THIS^.resetCycleManager();
configScope := THIS^.cycleManager.configuration;
THIS^.cycleManager.update(execute := TRUE);
AssertEquals_DINT(
	Expected := CNM_ReturnTypes.DefaultSteps.STEP.INIT,
	Actual := THIS^.cycleManager.step.current,
	Message := 'step should be INIT step'
);
// set global stepWidth
configScope.sequence.stepWidth := 7;
THIS^.cycleManager.proceed();
THIS^.cycleManager.update(execute := TRUE);
AssertEquals_DINT(
	Expected := (CNM_ReturnTypes.DefaultSteps.STEP.INIT + 7),
	Actual := THIS^.cycleManager.step.current,
	Message := 'step should be INIT step + 7'
);
// test it twice to make it nice
THIS^.cycleManager.proceed();
THIS^.cycleManager.update(execute := TRUE);
AssertEquals_DINT(
	Expected := (CNM_ReturnTypes.DefaultSteps.STEP.INIT + 14),
	Actual := THIS^.cycleManager.step.current,
	Message := 'step should be INIT step + 14'
);
// proceed with local stepWidth
THIS^.cycleManager.proceedWith(10);
THIS^.cycleManager.update(execute := TRUE);
AssertEquals_DINT(
	Expected := 10,
	Actual := THIS^.cycleManager.step.current,
	Message := 'stepWidth should be ignored by proceedWith(), step should be 10'
);
configScope.step.stepWidth := 5;
THIS^.cycleManager.proceed();
THIS^.cycleManager.update(execute := TRUE);
AssertEquals_DINT(
	Expected := 15,
	Actual := THIS^.cycleManager.step.current,
	Message := 'step should be 15'
);
// proceed again with global stepWidth
THIS^.cycleManager.proceed();
THIS^.cycleManager.update(execute := TRUE);
AssertEquals_DINT(
	Expected := 22,
	Actual := THIS^.cycleManager.step.current,
	Message := 'step should be 22'
);

TcUnit.TEST_FINISHED();
END_METHOD

(*

short summary
=================
Tests different stop request modes.
Verifies AFTER_SUCCESS, AFTER_NOT_SUCCESS, ALWAYS, and IGNORE modes work correctly.

.. <legal notes>

legal notes
=================
| SPDX-FileCopyrightText: © 2025 ekvip automation GmbH <info@ekvip.de>
| SPDX-License-Identifier: Apache-2.0
| For details check: Apache-2.0_

.. _Apache-2.0: https://www.apache.org/licenses/LICENSE-2.0

.. </legal notes>

*)
METHOD PRIVATE testStopRequestModes
VAR_INST
	testState : INT;
END_VAR
RETURN( THIS^.testSuiteAborted OR_ELSE  NOT TcUnit.TEST_ORDERED(THIS^.getTestNameFor('testStopRequestModes')));

CASE testState OF
0: // Initialize
	THIS^.resetCycleManager();
	iConfiguration := cycleManager;
	iCycleManager := cycleManager;
	testState := 10;
	
10: // Test AFTER_SUCCESS mode
	cycleManager.update(execute := TRUE, stopRequest := FALSE);
	
	// Configure stop request mode
	iConfiguration.configuration.sequence.stopRequest.afterSuccessfulStep();
	
	iCycleManager.proceedWith(10);
	cycleManager.update(execute := TRUE, stopRequest := FALSE);
	testState := 20;
	
20: // Evaluate success with stop request
	cycleManager.update(execute := TRUE, stopRequest := TRUE);
	AssertEquals_DINT(
		Expected := 10,
		Actual := iCycleManager.step.current,
		Message := 'Should stay in step 10 until successful evaluate'
	);
	IF iCycleManager.executeStep THEN
		// Evaluate success
		iCycleManager.evaluate(CNM_ReturnTypes.SingleExecutionState.SUCCESS);
		testState := 30;
	END_IF
	
30: // Verify moved to success due to stop request
	cycleManager.update(execute := TRUE, stopRequest := TRUE);
	
	AssertEquals_DINT(
		Expected := CNM_ReturnTypes.DefaultSteps.STEP.SUCCESS,
		Actual := iCycleManager.step.current,
		Message := 'Should move to SUCCESS with stop request after success'
	);
	
	AssertEquals_INT(
		Expected := CNM_ReturnTypes.SingleExecutionState.SUCCESS,
		Actual := iCycleManager.state,
		Message := 'state should be success after stop request'
	);
	
	// Test IGNORE mode
	cycleManager.update(execute := FALSE, stopRequest := FALSE);
	testState := 40;
	
40: // Test IGNORE mode
	cycleManager.update(execute := TRUE, stopRequest := FALSE);
	
	iConfiguration.configuration.sequence.stopRequest.ignore();
	
	iCycleManager.proceedWith(20);
	testState := 50;
	
50: // Stop request should be ignored
	cycleManager.update(execute := TRUE, stopRequest := TRUE);
	IF iCycleManager.executeStep THEN
		iCycleManager.evaluate(CNM_ReturnTypes.SingleExecutionState.SUCCESS);
		testState := 60;
	END_IF

60: // Verify proceeded normally
	cycleManager.update(execute := TRUE, stopRequest := TRUE);
	
	AssertEquals_DINT(
		Expected := 21, // Proceeded normally, not to SUCCESS
		Actual := iCycleManager.step.current,
		Message := 'Should proceed normally with IGNORE mode'
	);
	
	// Test ALWAYS mode
	cycleManager.update(execute := FALSE, stopRequest := FALSE);
	testState := 70;
	
70: // Test ALWAYS mode
	cycleManager.update(execute := TRUE, stopRequest := FALSE);
	
	iConfiguration.configuration.sequence.stopRequest.immediate();
	
	iCycleManager.proceedWith(30);
	cycleManager.update(execute := TRUE, stopRequest := FALSE);

	testState := 80;
	
80: // Stop request with ALWAYS mode
	cycleManager.update(execute := TRUE, stopRequest := TRUE);
	
	// Should immediately go to SUCCESS regardless of state
	testState := 90;
	
90: // Verify moved to SUCCESS
	cycleManager.update(execute := TRUE, stopRequest := TRUE);
	
	AssertEquals_DINT(
		Expected := CNM_ReturnTypes.DefaultSteps.STEP.SUCCESS,
		Actual := iCycleManager.step.current,
		Message := 'Should always move to SUCCESS with ALWAYS mode'
	);
	AssertEquals_INT(
		Expected := CNM_ReturnTypes.SingleExecutionState.SUCCESS,
		Actual := iCycleManager.state,
		Message := 'State should be SUCCESS'
	);
	
	// Test ALWAYS mode from error state
	cycleManager.update(execute := FALSE, stopRequest := FALSE);
	testState := 100;
	
100: // Setup for error state test
	cycleManager.update(execute := TRUE, stopRequest := FALSE);
	iCycleManager.proceedWith(40);
	testState := 110;
	
110: // Create error condition
	cycleManager.update(execute := TRUE, stopRequest := FALSE);
	IF iCycleManager.executeStep THEN
		iCycleManager.evaluate(
			state := CNM_ReturnTypes.SingleExecutionState.ERROR,
			errorStep := 999
		);
		testState := 120;
	END_IF
	
120: // In error step, activate stop request
	cycleManager.update(execute := TRUE, stopRequest := FALSE);
	AssertEquals_DINT(
		Expected := 999,
		Actual := iCycleManager.step.current,
		Message := 'Should be in error step'
	);
	cycleManager.update(execute := TRUE, stopRequest := TRUE);
	testState := 130;
	
130: // Verify ALWAYS mode works from error
	cycleManager.update(execute := TRUE, stopRequest := TRUE);
	AssertEquals_DINT(
		Expected := CNM_ReturnTypes.DefaultSteps.STEP.SUCCESS,
		Actual := iCycleManager.step.current,
		Message := 'ALWAYS mode should work even from error step'
	);
	
	// Test AFTER_NOT_SUCCESS mode
	cycleManager.update(execute := FALSE, stopRequest := FALSE);
	testState := 140;
	
140: // Test AFTER_NOT_SUCCESS mode
	cycleManager.update(execute := TRUE, stopRequest := FALSE);	
	iCycleManager.proceedWith(50);
	cycleManager.update(execute := TRUE, stopRequest := FALSE);
	cycleManager.update(execute := TRUE, stopRequest := FALSE);
	testState := 150;
	
150: // Evaluate SUCCESS with stop request
	iCycleManager.evaluate(CNM_ReturnTypes.SingleExecutionState.SUCCESS);
	iConfiguration.configuration.sequence.stopRequest.onBusy();
	cycleManager.update(execute := TRUE, stopRequest := TRUE);
	// With AFTER_NOT_SUCCESS and SUCCESS evaluation, should abort
	IF THIS^.cycleManager.executeStep THEN 
		testState := 160;
	END_IF
	
160: // Verify moved to step 51 instead of SUCCESS
	AssertEquals_DINT(
		Expected := 51,
		Actual := iCycleManager.step.current,
		Message := 'Should have moved to step 51'
	);
	
	// Test AFTER_NOT_SUCCESS with ERROR
	cycleManager.update(execute := FALSE, stopRequest := FALSE);
	cycleManager.update(execute := TRUE, stopRequest := FALSE);
	iCycleManager.proceedWith(60);
	testState := 170;
	
170: // Create error condition
	cycleManager.update(execute := TRUE, stopRequest := TRUE);
	iCycleManager.evaluate(
		state := CNM_ReturnTypes.SingleExecutionState.ERROR,
		errorStep := 888
	);
	IF iCycleManager.executeStep THEN
		testState := 180;
	END_IF
	
180: // Verify moved to SUCCESS after error
	cycleManager.update(execute := TRUE, stopRequest := TRUE);
	AssertEquals_DINT(
		Expected := 888,
		Actual := iCycleManager.step.current,
		Message := 'Should move to ERROR with ON_BUSY after ERROR'
	);
	
	// Test AFTER_NOT_SUCCESS with BUSY
	cycleManager.update(execute := FALSE, stopRequest := FALSE);
	testState := 190;
	
190: // Setup for error test
	cycleManager.update(execute := TRUE, stopRequest := FALSE);
	iCycleManager.proceedWith(70);
	testState := 200;
	
200: // Create error condition
	cycleManager.update(execute := TRUE, stopRequest := TRUE);
	iCycleManager.evaluate(
		state := CNM_ReturnTypes.SingleExecutionState.BUSY
	);
	IF iCycleManager.executeStep THEN
		testState := 210;
	END_IF
	
210: // Verify moved to SUCCESS after timeout
	cycleManager.update(execute := TRUE, stopRequest := TRUE);
	AssertEquals_DINT(
		Expected := CNM_ReturnTypes.DefaultSteps.STEP.SUCCESS,
		Actual := iCycleManager.step.current,
		Message := 'Should move to SUCCESS with AFTER_NOT_SUCCESS after BUSY'
	);
	
	cycleManager.update(execute := FALSE);
	testState := 0;
	TEST_FINISHED();
END_CASE
END_METHOD

(*

short summary
=================
Tests the succes step reuqired config. Normally the cyclemanager returns the state dependign on the current step (SUCCESS-Step = SUCCESS state).
To speed it up the SUCCESS state can be returned  on cycle earlier when transitioning to SUCCESS step.

.. <legal notes>

legal notes
=================
| SPDX-FileCopyrightText: © 2025 ekvip automation GmbH <info@ekvip.de>
| SPDX-License-Identifier: Apache-2.0
| For details check: Apache-2.0_

.. _Apache-2.0: https://www.apache.org/licenses/LICENSE-2.0

.. </legal notes>

*)

METHOD testSuccessRequiredConfig
VAR
	sequenceConfigScope :CNM_CycleManagerInterfaces.ISequenceConfiguration;
END_VAR
RETURN( THIS^.testSuiteAborted OR_ELSE  NOT TcUnit.TEST_ORDERED(THIS^.getTestNameFor('testSuccessRequiredConfig')));

THIS^.resetCycleManager();
sequenceConfigScope := cycleManager.configuration.sequence;
cycleManager.update(execute := TRUE);
cycleManager.update(execute := TRUE);
sequenceConfigScope.requireSuccessStep := TRUE;
cycleManager.step.next := CNM_ReturnTypes.DefaultSteps.STEP.SUCCESS;
cycleManager.evaluate(state := CNM_ReturnTypes.SingleExecutionState.SUCCESS);
AssertEquals_DINT(
	Expected := CNM_ReturnTypes.DefaultSteps.STEP.INIT,
	Actual := THIS^.cycleManager.step.current,
	Message := 'Step should be INIT'
);
AssertEquals_INT(
	Expected := CNM_ReturnTypes.SingleExecutionState.BUSY,
	Actual := cycleManager.state,
	Message := 'State should be busy'
); 
cycleManager.update(execute := TRUE);
AssertEquals_DINT(
	Expected := CNM_ReturnTypes.DefaultSteps.STEP.SUCCESS,
	Actual := THIS^.cycleManager.step.current,
	Message := 'Step should be SUCCESS'
);
AssertEquals_INT(
	Expected := CNM_ReturnTypes.SingleExecutionState.SUCCESS,
	Actual := cycleManager.state,
	Message := 'State should be SUCCESS'
);
	
cycleManager.update(execute := FALSE);
cycleManager.update(execute := TRUE);
cycleManager.update(execute := TRUE);
sequenceConfigScope.requireSuccessStep := FALSE;
cycleManager.step.next := CNM_ReturnTypes.DefaultSteps.STEP.SUCCESS;
cycleManager.evaluate(state := CNM_ReturnTypes.SingleExecutionState.SUCCESS);
AssertEquals_DINT(
	Expected := CNM_ReturnTypes.DefaultSteps.STEP.INIT,
	Actual := THIS^.cycleManager.step.current,
	Message := 'Step should be INIT'
);
AssertEquals_INT(
	Expected := CNM_ReturnTypes.SingleExecutionState.SUCCESS,
	Actual := cycleManager.state,
	Message := 'State should be SUCCESS immediately '
);

TcUnit.TEST_FINISHED();
END_METHOD

(*

short summary
=================
Tests timeout behavior of the cycle manager.
Verifies timeout configuration and automatic transition to timeout step.

.. <legal notes>

legal notes
=================
| SPDX-FileCopyrightText: © 2025 ekvip automation GmbH <info@ekvip.de>
| SPDX-License-Identifier: Apache-2.0
| For details check: Apache-2.0_

.. _Apache-2.0: https://www.apache.org/licenses/LICENSE-2.0

.. </legal notes>

*)
METHOD PRIVATE testTimeoutBehavior
VAR_INST
	testState : INT;
	timeoutTimer : TON;
END_VAR
RETURN( THIS^.testSuiteAborted OR_ELSE  NOT TcUnit.TEST_ORDERED(THIS^.getTestNameFor('testTimeoutBehavior')));

CASE testState OF
0: // Initialize
	THIS^.resetCycleManager();
	iConfiguration := cycleManager;
	iCycleManager := cycleManager;
	testState := 10;
	
10: // Configure timeout
	cycleManager.update(execute := TRUE);
	
	// Set sequence timeout
	iConfiguration.configuration.sequence.timeout := T#100MS;
	iConfiguration.configuration.sequence.timeoutStep := 999;
	
	iCycleManager.proceedWith(10);
	testState := 20;
	
20: // Wait for timeout
	cycleManager.update(execute := TRUE); // Disable step control to trigger timeout
	// Start timer to track timeout
	timeoutTimer(IN := cycleManager.executeStep, PT := T#110MS);
	CASE cycleManager.step.current OF 
	10:
		IF timeoutTimer.Q THEN
			AssertTrue(
				Condition := FALSE,
				Message := 'Cyclemanager timeout not triggered in time'
			);
			testState := 100;
		END_IF
	999:
		testState := 30;
	ELSE
		AssertTrue(
			Condition := FALSE,
			Message := 'wrong step after timeout monitoring detected'
		);
		testState := 100;
	END_CASE
	
30:
	AssertTrue(
		Condition := cycleManager.errors.isInErrorStep,
		Message := 'Timeout step should be marked as error step'
	);
	cycleManager.proceedWith(10);
	testState := 40;
40:
	cycleManager.update(execute := TRUE);
	cycleManager.configuration.step.timeoutStep := 666;
	cycleManager.configuration.step.timeout := T#50MS;
	timeoutTimer(IN := cycleManager.executeStep, PT := T#60MS);
	CASE cycleManager.step.current OF
	10:
		IF timeoutTimer.Q THEN
			AssertTrue(
				Condition := FALSE,
				Message := 'Cyclemanager timeout not triggered in time'
			);
			testState := 100;
		END_IF
	666:
		testState := 50;
		AssertTrue(
			Condition := cycleManager.errors.isInErrorStep,
			Message := 'Timeout step should be marked as error step'
		);
		cycleManager.proceedWith(10);	
	999:
		AssertTrue(
			Condition := FALSE,
			Message := 'global sequence timeout triggered instead of local step configuration'
		);
		testState := 100;
	ELSE
		AssertTrue(
			Condition := FALSE,
			Message := 'wrong step after timeout monitoring detected'
		);
		testState := 100;	
	END_CASE
50:
	// Wait for timeout
	cycleManager.update(execute := TRUE); // Disable step control to trigger timeout
	// Start timer to track timeout
	timeoutTimer(IN := cycleManager.executeStep, PT := T#110MS);
	CASE cycleManager.step.current OF 
	10:
		IF timeoutTimer.Q THEN
			AssertTrue(
				Condition := FALSE,
				Message := 'Cyclemanager timeout not triggered in time'
			);
			testState := 100;
		END_IF
	999:
		testState := 100;
	ELSE
		AssertTrue(
			Condition := FALSE,
			Message := 'wrong step after timeout monitoring detected'
		);
		testState := 100;
	END_CASE
100:
	TEST_FINISHED();
END_CASE
END_METHOD

(*

short summary
=================
Tests the waitFor() method behavior.
Verifies that the cycle manager waits for a boolean condition before proceeding.

.. <legal notes>

legal notes
=================
| SPDX-FileCopyrightText: © 2025 ekvip automation GmbH <info@ekvip.de>
| SPDX-License-Identifier: Apache-2.0
| For details check: Apache-2.0_

.. _Apache-2.0: https://www.apache.org/licenses/LICENSE-2.0

.. </legal notes>

*)
METHOD PRIVATE testWaitForMethod
VAR_INST
	testState : INT;
	waitCondition : BOOL;
	cycleCount : INT;
END_VAR
VAR
	foo :POINTER TO BYTE := ADR(waitCondition);
	bar : ARRAY [0..1] OF DINT := [10, 11];
	
END_VAR
RETURN( THIS^.testSuiteAborted OR_ELSE  NOT TcUnit.TEST_ORDERED(THIS^.getTestNameFor('testWaitForMethod')));

CASE testState OF
0: // Initialize
	THIS^.resetCycleManager();
	iCycleManager := cycleManager;
	waitCondition := FALSE;
	cycleCount := 0;
	testState := 10;
	
10: // Start and move to test step
	cycleManager.update(execute := TRUE);
	iCycleManager.proceedWith(10);
	testState := 20;
	cycleManager.update(execute := TRUE);
	
20: // Test waitFor
	// After 3 cycles, set condition true
	cycleCount := cycleCount + 1;
	IF cycleCount >= 4 THEN
		waitCondition := TRUE;
		testState := 30;
		cycleCount := 0;
	END_IF
	iCycleManager.waitFor(value := waitCondition);
	
	cycleManager.update(execute := TRUE);
	// Wait should keep step busy
	AssertEquals_DINT(
		Expected := bar[foo^],
		Actual := iCycleManager.step.current,
		Message := 'Step should only change when waitForCondition is true'
	);
	waitCondition := FALSE;
	
30: // Verify proceeded to next step
	cycleManager.update(execute := TRUE);
	cycleManager.waitFor(TRUE);
	AssertEquals_DINT(
		Expected := 11, // Default step width is 1
		Actual := iCycleManager.step.current,
		Message := 'Should not proceed without update call'
	);
	cycleManager.update(execute := TRUE);
	AssertEquals_DINT(
		Expected := 12, // Default step width is 1
		Actual := iCycleManager.step.current,
		Message := 'Should proceed after update call'
	);
	
	TEST_FINISHED();	
END_CASE
END_METHOD

END_FUNCTION_BLOCK

// ---- Project Information/F_GetCompany.TcPOU
// This function has been automatically generated from the project information.
{attribute 'signature_flag' := '1073741824'}
{attribute 'TcGenerated'}
{attribute 'no-analysis'}
FUNCTION F_GetCompany : WSTRING
VAR_INPUT
	
END_VAR

F_GetCompany := "ekvip automation GmbH";

END_FUNCTION

// ---- Project Information/F_GetTitle.TcPOU
// This function has been automatically generated from the project information.
{attribute 'signature_flag' := '1073741824'}
{attribute 'TcGenerated'}
{attribute 'no-analysis'}
FUNCTION F_GetTitle : WSTRING
VAR_INPUT
	
END_VAR

F_GetTitle := "CNM_CycleManagerInterfacesTests";

END_FUNCTION

// ---- Project Information/F_GetVersion.TcPOU
// This function has been automatically generated from the project information.
{attribute 'signature_flag' := '1073741824'}
{attribute 'TcGenerated'}
{attribute 'no-analysis'}
FUNCTION F_GetVersion : ST_LibVersion
VAR_INPUT
	
END_VAR

F_GetVersion.iMajor := 1;
F_GetVersion.iMinor := 0;
F_GetVersion.iBuild := 0;
F_GetVersion.iRevision := 0;
F_GetVersion.sVersion := '1.0.0.0';
F_GetVersion.nFlags := 0;

END_FUNCTION
